PROGRAM Controls_MAIN
VAR
END_VAR


//Aliohjelmiesn kutsuja läjä tänne

END_PROGRAM

(* stored: Version 1.1.0.1, ProductVersion 3.1.4024.10
   POU Controls_MAIN: Id {27560784-429a-4cb9-b530-4b903427c533}, SpecialFunc None *)
